(* Logix 5000 project; controller cal1615 1756-L62 rev 20.11; software revision 20.05; part 29 of 82 *)
(* tags used below, declared in another part *)
   FAULT : BOOL;   // Fault AFI
   HMI : BOOL;   // AFI HMI
   p01_sys_scp : SYS_SCP;   // System Scaling
   p01r02 : routine;   // System Misc Control
   p01r09_pb_global_reset : BOOL;   // System Modes PB: Global Fault Reset
   p13_ai_exhaust_amps : REAL;   // Zone 3 Analog Input Exhaust Fan Amps
   p13_ai_exhaust_hz : REAL;   // Zone 3 Analog Input Exhaust Fan HZ
   p13_ai_exhaust_hz_max : REAL;   // Zone 3 Analog Input Exhaust Fan Max HZ
   p13_ai_exhaust_rpm : REAL;   // Zone 3 Analog Input Exhaust Fan RPM
   p13_ai_recirc_amps : REAL;   // Zone 3 Analog Input Recirc Fan Amps
   p13_ai_recirc_hz : REAL;   // Zone 3 Analog Input Supply Fan HZ
   p13_ai_recirc_hz_max : REAL;   // Zone 3 Analog Input Supply Fan max HZ
   p13_ai_recirc_rpm : REAL;   // Zone 3 Analog Input Recirc Fan RPM
   p13_ai_tc01 : REAL;   // Zone 3 Analog Input Control Thermocouple 1
   p13_ai_tc02 : REAL;   // Zone 3 Analog Input Control Thermocouple 2
   p13_ao_cv : REAL;   // Zone 3 Analog Output Control Valve
   p13_ao_exhaust_selected_speed : REAL;   // Zone 3 Analog Output Exhaust Fan VFD Selected Speed
   p13_ao_recirc_selected_speed : REAL;   // Zone 3 Analog Output Recirc Fan VFD Selected Speed
   p13_di_door_open : BOOL;   // Zone 3 Digital Input Access Door Open
   p13_di_exh : acs800_di_normal;   // Zone 3 Digital Inputs Exhaust Fan
   p13_di_exh_fan_mtr_ts : BOOL;   // Zone 3 Digital Input Exhaust Fan Motor Thermostat OK
   p13_di_exh_flow_ok : BOOL;   // Zone 3 Digital Input Exhaust Flow OK
   p13_di_filter_clean : BOOL;   // Zone 3 Digital Input Filter Dirty
   p13_di_recirc : acs800_di_normal;   // Zone 3 Digital Inputs Recirc Fan
   p13_di_recirc_fan_mtr_ts : BOOL;   // Zone 3 Digital Input Recirc Fan Motor Thermostat OK
   p13_di_recirc_flow_ok : BOOL;   // Zone 3 Digital Input Recirc Flow OK
   p13_di_tc01_bo : BOOL;   // Zone 3 Digital Input Control Thermocouple 1 Failure
   p13_di_tc02_bo : BOOL;   // Zone 3 Digital Input Control Thermocouple 2 Failure
   p13_dint_to_hmi : DINT[16];   // Zone 3 Temperature Control VFDs On
   p13_do_exh : acs800_do_normal;   // Zone 3 Digital Output Exhaust Fan
   p13_do_recirc : acs800_do_normal;   // Zone 3 Digital Outputs Supply Fan
   p13_exhaust_input_max : REAL;
   p13_exhaust_input_min : REAL;
   p13_exhaust_output_max : REAL;
   p13_exhaust_output_min : REAL;
   p13_hc_input_max : REAL;
   p13_hc_input_min : REAL;
   p13_hc_output_max : REAL;
   p13_hc_output_min : REAL;
   p13_param_tc01z : REAL;   // Zone 3 Parameter Process Temperature Zero Offset
   p13_param_tc02z : REAL;   // Zone 3 Parameter SupplyTemperature Zero Offset
   p13_recirc_input_max : REAL;
   p13_recirc_input_min : REAL;
   p13_recirc_output_max : REAL;
   p13_recirc_output_min : REAL;
   p13r01 : routine;   // Zone 3 Main
   p13r03 : routine;   // Zone 3 Input
   p13r03_hz : SYS_SCP;   // Zone 3 Analog Inputs SCP Hz
   p13r03_timer_fault : TIMER[4];   // Zone 3 Input Fault Delay
   p13r03_timer_warning : TIMER[4];   // Zone 3 Input Warning Delay
   p13r04 : routine;   // Zone 3 Output
   p13r04_timer_fault : TIMER[4];   // Zone 3 Output Fault Delay
   p13r04_timer_warning : TIMER[4];   // Zone 3 Output Warning Delay
   p13r05 : routine;   // Zone 3 Dint to HMI
   p13r05_exh_status : DINT;
   p13r05_temp_ctl_status : DINT;
   p13r20_state : DINT;   // Zone 3 Temperature Control State
   p13r20_status : DINT;   // Zone 3 Temperature Control Sequence Status
   p13r30 : routine;   // Zone 3 Temperature Control
   p13r30_permissive_run : BOOL;   // Zone 3 Temperature Control Run Permissive
   p13r30_request_cool : BOOL;   // Zone 3 Temperature Control Request Cooling
   p13r30_request_manual : BOOL;   // Zone 3 Temperature Control Request Manual Control
   p13r30_vfds_ready : BOOL;   // Zone 3 Temperature Control VFDs On
   p13r31 : routine;   // Zone 3 Exhaust VFD
   p13r31_request_auto_run : BOOL;   // Zone 3 Exhaust Fan Run Request
   p13r31_request_auto_stop : BOOL;   // Zone 3 Exhaust VFD Request Auto Stop
   p13r31_vfd_stopped : BOOL;   // Zone 3 Exhaust VFD VFD Stopped
   p13r32_request_auto_run : BOOL;   // Zone 3 Recirc Fan Run Request
   p13r32_request_auto_stop : BOOL;   // Zone 3 Recirc VFD Request Auto Stop
(* P13_Zone_3, continued *)

ROUTINE R03_Input   (* ladder *)
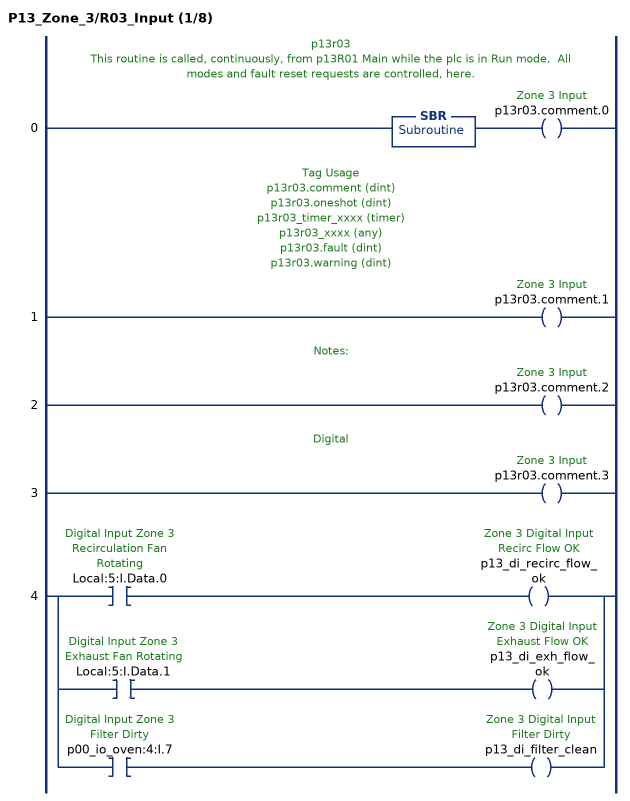
   // p13r03
   // This routine is called, continuously, from p13R01 Main while the plc is in Run mode.  All modes and fault reset requests are controlled, here.
   0: SBR()OTE(p13r03.comment.0);
   // Tag Usage
   // p13r03.comment (dint)
   // p13r03.oneshot (dint)
   // p13r03_timer_xxxx (timer)
   // p13r03_xxxx (any)
   // p13r03.fault (dint)
   // p13r03.warning (dint)
   1: OTE(p13r03.comment.1);
   // Notes:
   2: OTE(p13r03.comment.2);
   // Digital
   3: OTE(p13r03.comment.3);
   4: [XIC(Local:5:I.Data.0) OTE(p13_di_recirc_flow_ok) ,XIC(Local:5:I.Data.1) OTE(p13_di_exh_flow_ok) ,XIC(p00_io_oven:4:I.7) OTE(p13_di_filter_clean) ];
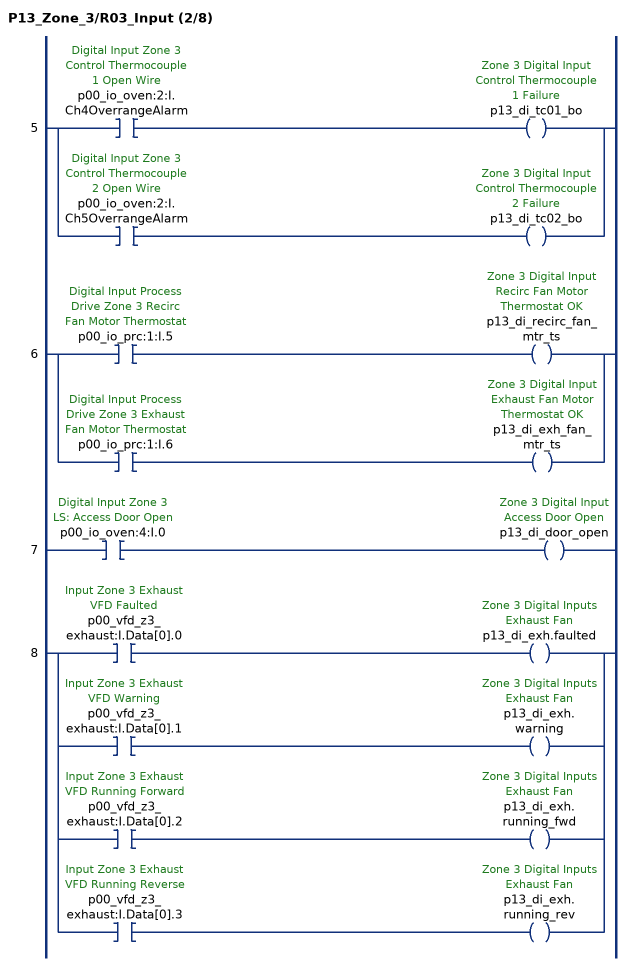
   5: [XIC(p00_io_oven:2:I.Ch4OverrangeAlarm) OTE(p13_di_tc01_bo) ,XIC(p00_io_oven:2:I.Ch5OverrangeAlarm) OTE(p13_di_tc02_bo) ];
   6: [XIC(p00_io_prc:1:I.5) OTE(p13_di_recirc_fan_mtr_ts) ,XIC(p00_io_prc:1:I.6) OTE(p13_di_exh_fan_mtr_ts) ];
   7: XIC(p00_io_oven:4:I.0)OTE(p13_di_door_open);
   8: [XIC(p00_vfd_z3_exhaust:I.Data[0].0) OTE(p13_di_exh.faulted) ,XIC(p00_vfd_z3_exhaust:I.Data[0].1) OTE(p13_di_exh.warning) ,XIC(p00_vfd_z3_exhaust:I.Data[0].2) OTE(p13_di_exh.running_fwd) ,XIC(p00_vfd_z3_exhaust:I.Data[0].3) OTE(p13_di_exh.running_rev) ];
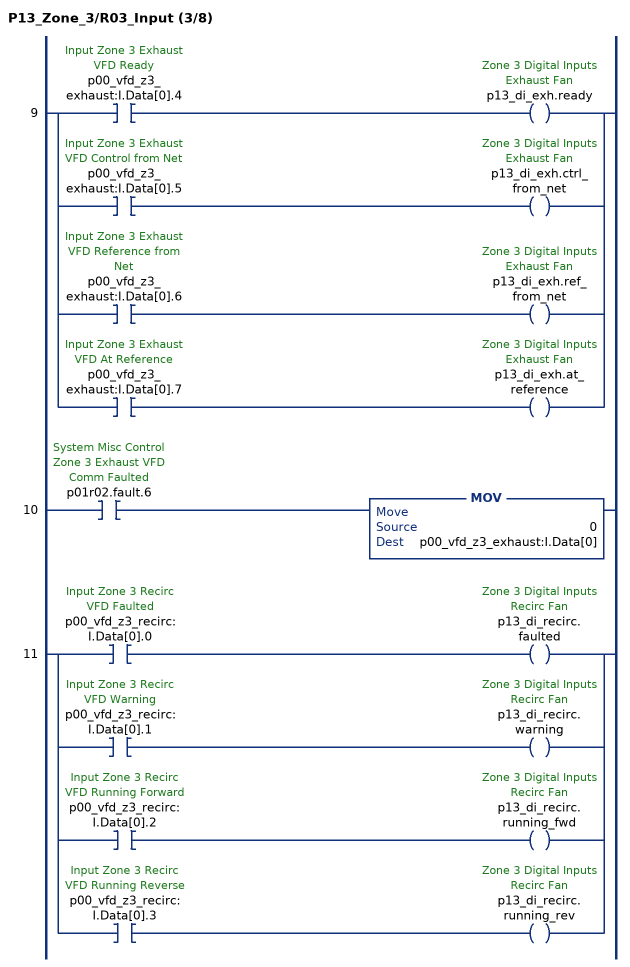
   9: [XIC(p00_vfd_z3_exhaust:I.Data[0].4) OTE(p13_di_exh.ready) ,XIC(p00_vfd_z3_exhaust:I.Data[0].5) OTE(p13_di_exh.ctrl_from_net) ,XIC(p00_vfd_z3_exhaust:I.Data[0].6) OTE(p13_di_exh.ref_from_net) ,XIC(p00_vfd_z3_exhaust:I.Data[0].7) OTE(p13_di_exh.at_reference) ];
   10: XIC(p01r02.fault.6)MOV(0,p00_vfd_z3_exhaust:I.Data[0]);
   11: [XIC(p00_vfd_z3_recirc:I.Data[0].0) OTE(p13_di_recirc.faulted) ,XIC(p00_vfd_z3_recirc:I.Data[0].1) OTE(p13_di_recirc.warning) ,XIC(p00_vfd_z3_recirc:I.Data[0].2) OTE(p13_di_recirc.running_fwd) ,XIC(p00_vfd_z3_recirc:I.Data[0].3) OTE(p13_di_recirc.running_rev) ];
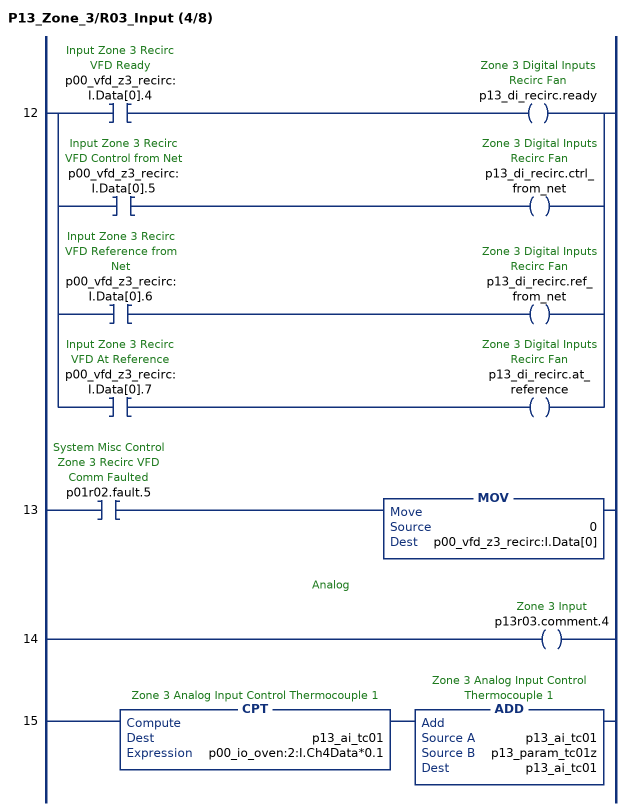
   12: [XIC(p00_vfd_z3_recirc:I.Data[0].4) OTE(p13_di_recirc.ready) ,XIC(p00_vfd_z3_recirc:I.Data[0].5) OTE(p13_di_recirc.ctrl_from_net) ,XIC(p00_vfd_z3_recirc:I.Data[0].6) OTE(p13_di_recirc.ref_from_net) ,XIC(p00_vfd_z3_recirc:I.Data[0].7) OTE(p13_di_recirc.at_reference) ];
   13: XIC(p01r02.fault.5)MOV(0,p00_vfd_z3_recirc:I.Data[0]);
   // Analog
   14: OTE(p13r03.comment.4);
   15: CPT(p13_ai_tc01,p00_io_oven:2:I.Ch4Data*0.1)ADD(p13_ai_tc01,p13_param_tc01z,p13_ai_tc01);
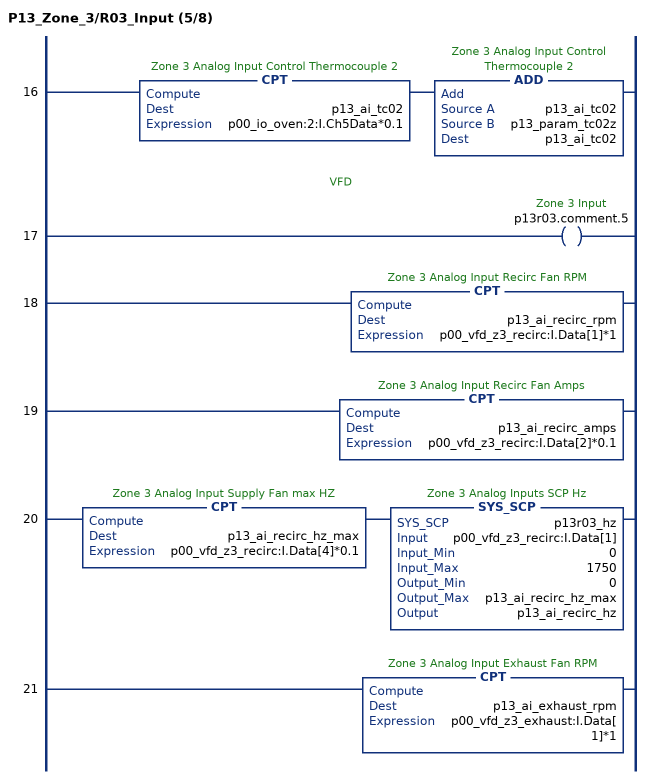
   16: CPT(p13_ai_tc02,p00_io_oven:2:I.Ch5Data*0.1)ADD(p13_ai_tc02,p13_param_tc02z,p13_ai_tc02);
   // VFD
   17: OTE(p13r03.comment.5);
   18: CPT(p13_ai_recirc_rpm,p00_vfd_z3_recirc:I.Data[1]*1);
   19: CPT(p13_ai_recirc_amps,p00_vfd_z3_recirc:I.Data[2]*0.1);
   20: CPT(p13_ai_recirc_hz_max,p00_vfd_z3_recirc:I.Data[4]*0.1)SYS_SCP(p13r03_hz,p00_vfd_z3_recirc:I.Data[1],0,1750,0,p13_ai_recirc_hz_max,p13_ai_recirc_hz);
   21: CPT(p13_ai_exhaust_rpm,p00_vfd_z3_exhaust:I.Data[1]*1);
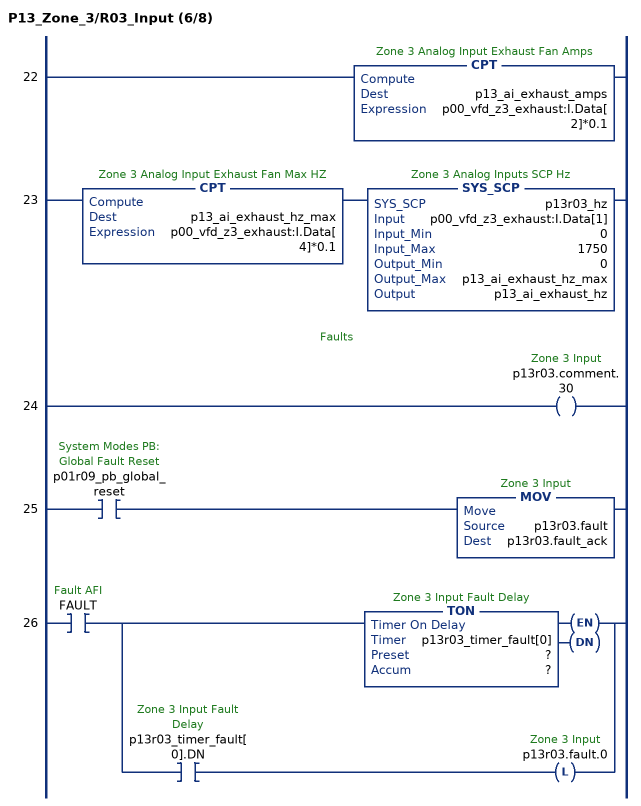
   22: CPT(p13_ai_exhaust_amps,p00_vfd_z3_exhaust:I.Data[2]*0.1);
   23: CPT(p13_ai_exhaust_hz_max,p00_vfd_z3_exhaust:I.Data[4]*0.1)SYS_SCP(p13r03_hz,p00_vfd_z3_exhaust:I.Data[1],0,1750,0,p13_ai_exhaust_hz_max,p13_ai_exhaust_hz);
   // Faults
   24: OTE(p13r03.comment.30);
   25: XIC(p01r09_pb_global_reset)MOV(p13r03.fault,p13r03.fault_ack);
   26: XIC(FAULT)[TON(p13r03_timer_fault[0],?,?) ,XIC(p13r03_timer_fault[0].DN) OTL(p13r03.fault.0) ];
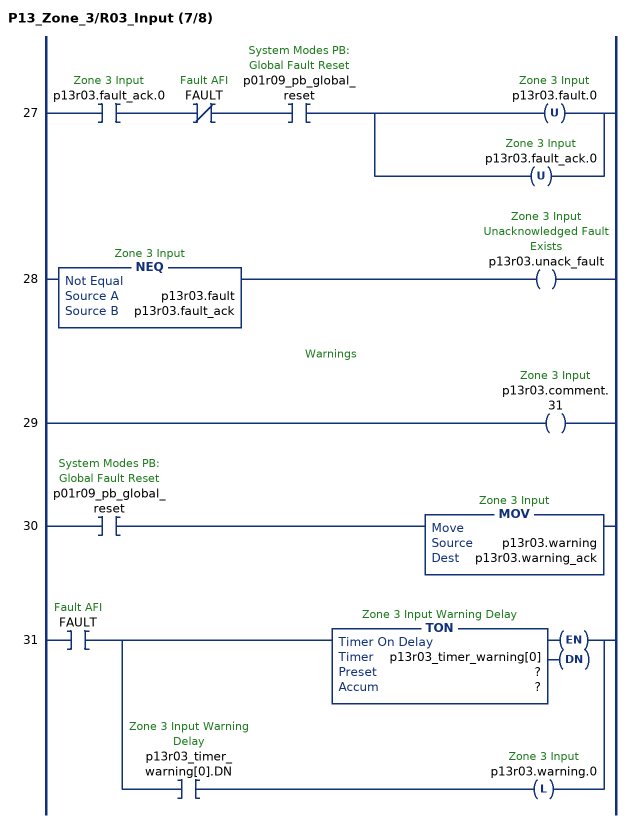
   27: XIC(p13r03.fault_ack.0)XIO(FAULT)XIC(p01r09_pb_global_reset)[OTU(p13r03.fault.0) ,OTU(p13r03.fault_ack.0) ];
   28: NEQ(p13r03.fault,p13r03.fault_ack)OTE(p13r03.unack_fault);
   // Warnings
   29: OTE(p13r03.comment.31);
   30: XIC(p01r09_pb_global_reset)MOV(p13r03.warning,p13r03.warning_ack);
   31: XIC(FAULT)[TON(p13r03_timer_warning[0],?,?) ,XIC(p13r03_timer_warning[0].DN) OTL(p13r03.warning.0) ];
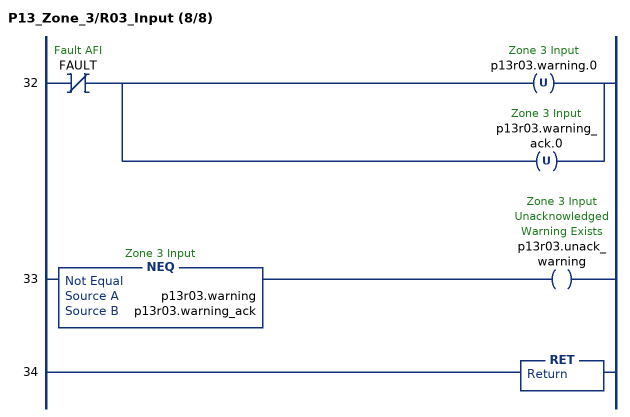
   32: XIO(FAULT)[OTU(p13r03.warning.0) ,OTU(p13r03.warning_ack.0) ];
   33: NEQ(p13r03.warning,p13r03.warning_ack)OTE(p13r03.unack_warning);
   34: RET();
END_ROUTINE

ROUTINE R04_Output   (* ladder *)
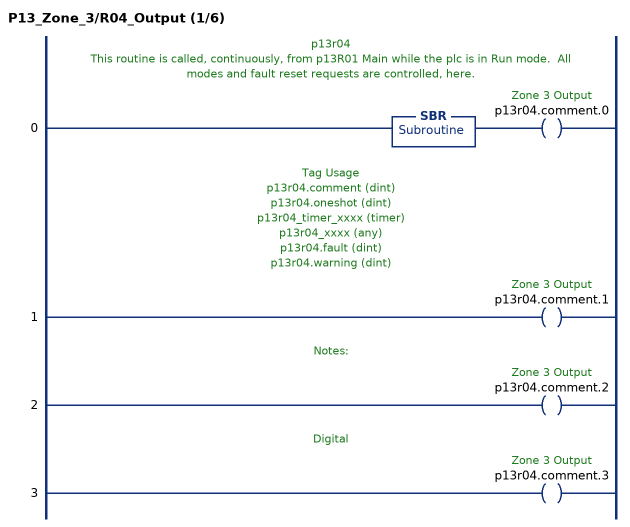
   // p13r04
   // This routine is called, continuously, from p13R01 Main while the plc is in Run mode.  All modes and fault reset requests are controlled, here.
   0: SBR()OTE(p13r04.comment.0);
   // Tag Usage
   // p13r04.comment (dint)
   // p13r04.oneshot (dint)
   // p13r04_timer_xxxx (timer)
   // p13r04_xxxx (any)
   // p13r04.fault (dint)
   // p13r04.warning (dint)
   1: OTE(p13r04.comment.1);
   // Notes:
   2: OTE(p13r04.comment.2);
   // Digital
   3: OTE(p13r04.comment.3);
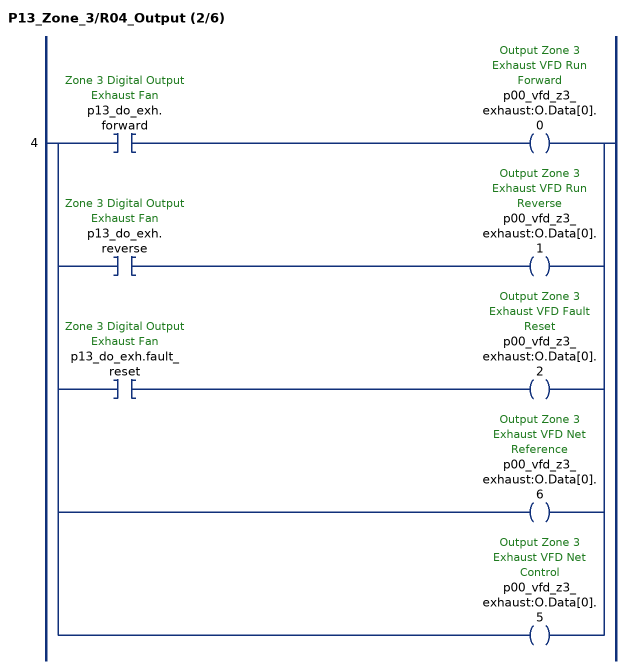
   4: [XIC(p13_do_exh.forward) OTE(p00_vfd_z3_exhaust:O.Data[0].0) ,XIC(p13_do_exh.reverse) OTE(p00_vfd_z3_exhaust:O.Data[0].1) ,XIC(p13_do_exh.fault_reset) OTE(p00_vfd_z3_exhaust:O.Data[0].2) ,OTE(p00_vfd_z3_exhaust:O.Data[0].6) ,OTE(p00_vfd_z3_exhaust:O.Data[0].5) ];
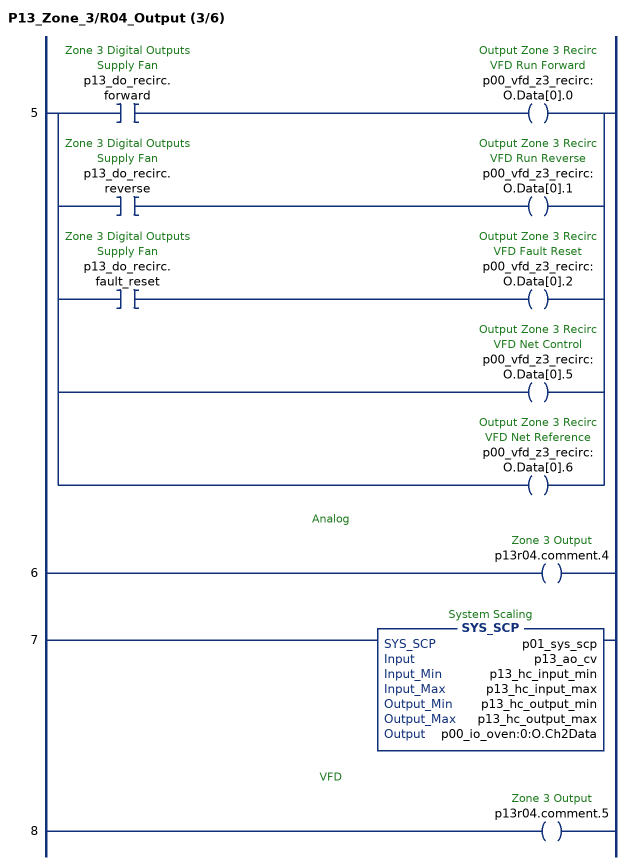
   5: [XIC(p13_do_recirc.forward) OTE(p00_vfd_z3_recirc:O.Data[0].0) ,XIC(p13_do_recirc.reverse) OTE(p00_vfd_z3_recirc:O.Data[0].1) ,XIC(p13_do_recirc.fault_reset) OTE(p00_vfd_z3_recirc:O.Data[0].2) ,OTE(p00_vfd_z3_recirc:O.Data[0].5) ,OTE(p00_vfd_z3_recirc:O.Data[0].6) ];
   // Analog
   6: OTE(p13r04.comment.4);
   7: SYS_SCP(p01_sys_scp,p13_ao_cv,p13_hc_input_min,p13_hc_input_max,p13_hc_output_min,p13_hc_output_max,p00_io_oven:0:O.Ch2Data);
   // VFD
   8: OTE(p13r04.comment.5);
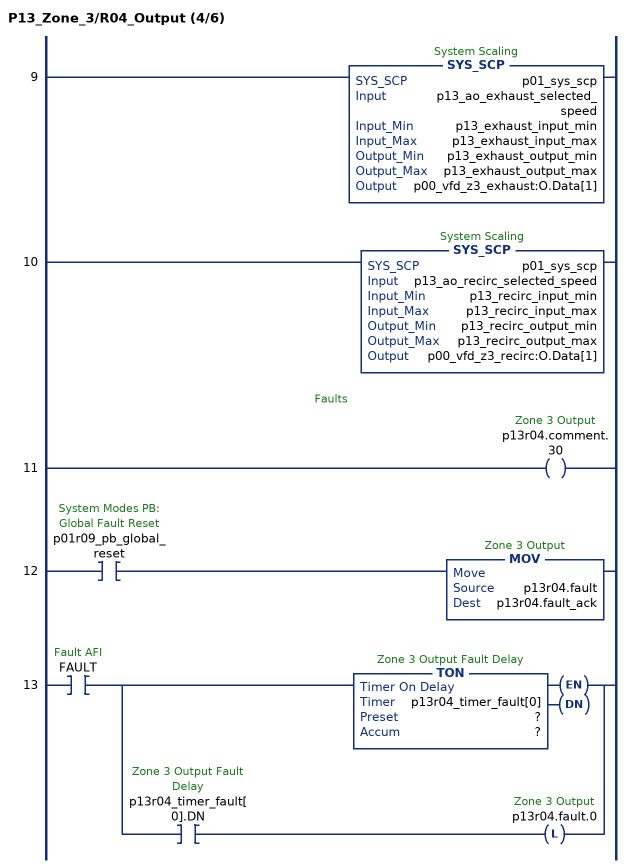
   9: SYS_SCP(p01_sys_scp,p13_ao_exhaust_selected_speed,p13_exhaust_input_min,p13_exhaust_input_max,p13_exhaust_output_min,p13_exhaust_output_max,p00_vfd_z3_exhaust:O.Data[1]);
   10: SYS_SCP(p01_sys_scp,p13_ao_recirc_selected_speed,p13_recirc_input_min,p13_recirc_input_max,p13_recirc_output_min,p13_recirc_output_max,p00_vfd_z3_recirc:O.Data[1]);
   // Faults
   11: OTE(p13r04.comment.30);
   12: XIC(p01r09_pb_global_reset)MOV(p13r04.fault,p13r04.fault_ack);
   13: XIC(FAULT)[TON(p13r04_timer_fault[0],?,?) ,XIC(p13r04_timer_fault[0].DN) OTL(p13r04.fault.0) ];
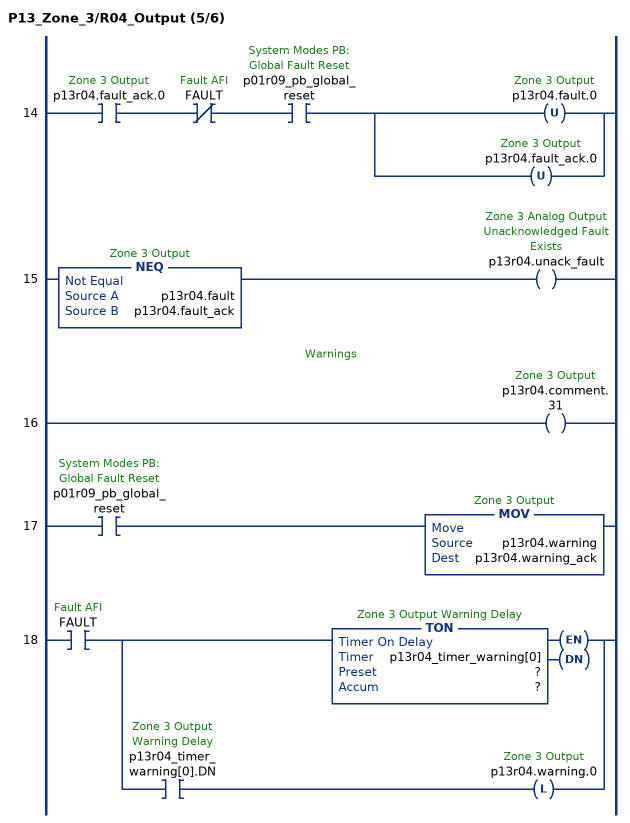
   14: XIC(p13r04.fault_ack.0)XIO(FAULT)XIC(p01r09_pb_global_reset)[OTU(p13r04.fault.0) ,OTU(p13r04.fault_ack.0) ];
   15: NEQ(p13r04.fault,p13r04.fault_ack)OTE(p13r04.unack_fault);
   // Warnings
   16: OTE(p13r04.comment.31);
   17: XIC(p01r09_pb_global_reset)MOV(p13r04.warning,p13r04.warning_ack);
   18: XIC(FAULT)[TON(p13r04_timer_warning[0],?,?) ,XIC(p13r04_timer_warning[0].DN) OTL(p13r04.warning.0) ];
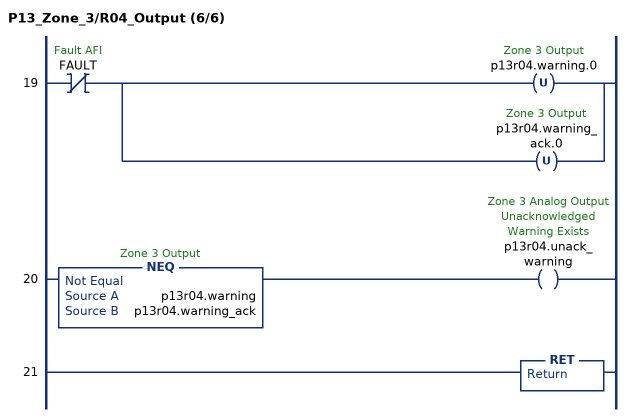
   19: XIO(FAULT)[OTU(p13r04.warning.0) ,OTU(p13r04.warning_ack.0) ];
   20: NEQ(p13r04.warning,p13r04.warning_ack)OTE(p13r04.unack_warning);
   21: RET();
END_ROUTINE

ROUTINE R05_Dint_to_HMI   (* ladder *)
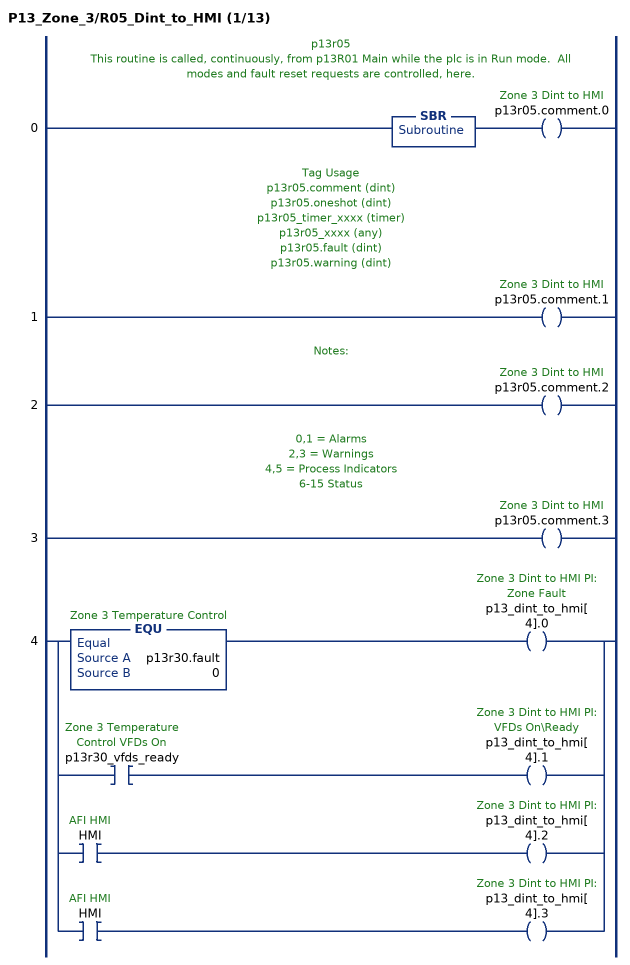
   // p13r05
   // This routine is called, continuously, from p13R01 Main while the plc is in Run mode.  All modes and fault reset requests are controlled, here.
   0: SBR()OTE(p13r05.comment.0);
   // Tag Usage
   // p13r05.comment (dint)
   // p13r05.oneshot (dint)
   // p13r05_timer_xxxx (timer)
   // p13r05_xxxx (any)
   // p13r05.fault (dint)
   // p13r05.warning (dint)
   1: OTE(p13r05.comment.1);
   // Notes:
   2: OTE(p13r05.comment.2);
   // 0,1 = Alarms
   // 2,3 = Warnings
   // 4,5 = Process Indicators
   // 6-15 Status
   3: OTE(p13r05.comment.3);
   4: [EQU(p13r30.fault,0) OTE(p13_dint_to_hmi[4].0) ,XIC(p13r30_vfds_ready) OTE(p13_dint_to_hmi[4].1) ,XIC(HMI) OTE(p13_dint_to_hmi[4].2) ,XIC(HMI) OTE(p13_dint_to_hmi[4].3) ];
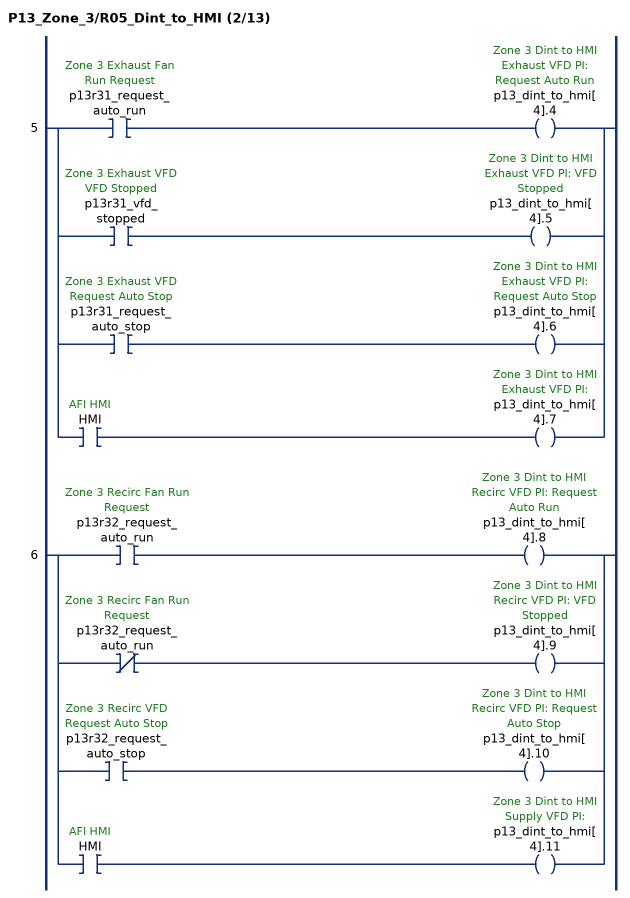
   5: [XIC(p13r31_request_auto_run) OTE(p13_dint_to_hmi[4].4) ,XIC(p13r31_vfd_stopped) OTE(p13_dint_to_hmi[4].5) ,XIC(p13r31_request_auto_stop) OTE(p13_dint_to_hmi[4].6) ,XIC(HMI) OTE(p13_dint_to_hmi[4].7) ];
   6: [XIC(p13r32_request_auto_run) OTE(p13_dint_to_hmi[4].8) ,XIO(p13r32_request_auto_run) OTE(p13_dint_to_hmi[4].9) ,XIC(p13r32_request_auto_stop) OTE(p13_dint_to_hmi[4].10) ,XIC(HMI) OTE(p13_dint_to_hmi[4].11) ];
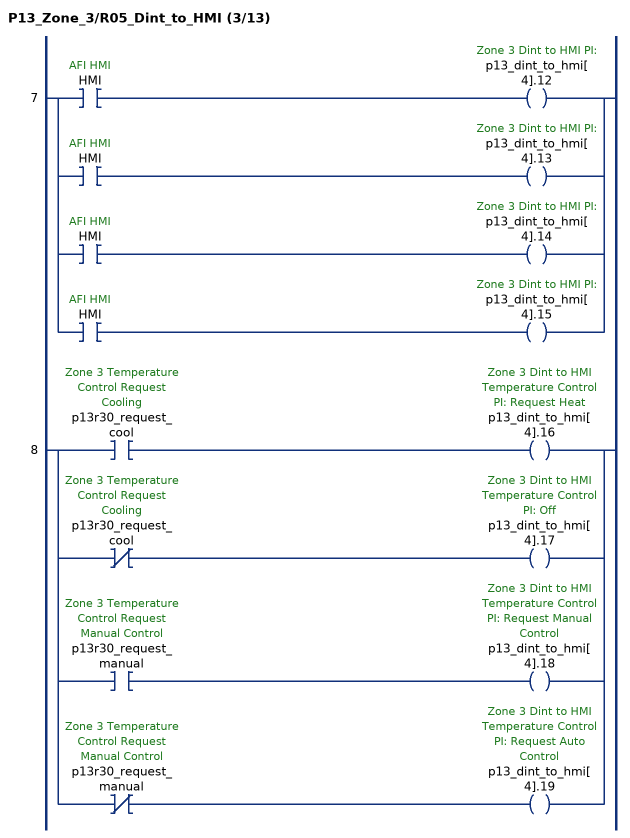
   7: [XIC(HMI) OTE(p13_dint_to_hmi[4].12) ,XIC(HMI) OTE(p13_dint_to_hmi[4].13) ,XIC(HMI) OTE(p13_dint_to_hmi[4].14) ,XIC(HMI) OTE(p13_dint_to_hmi[4].15) ];
   8: [XIC(p13r30_request_cool) OTE(p13_dint_to_hmi[4].16) ,XIO(p13r30_request_cool) OTE(p13_dint_to_hmi[4].17) ,XIC(p13r30_request_manual) OTE(p13_dint_to_hmi[4].18) ,XIO(p13r30_request_manual) OTE(p13_dint_to_hmi[4].19) ];
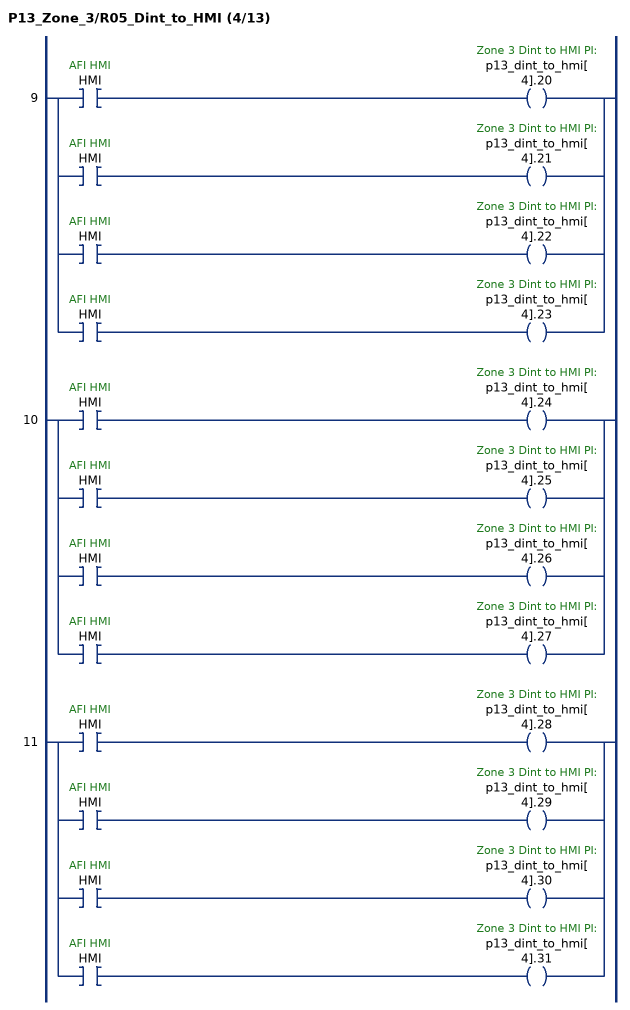
   9: [XIC(HMI) OTE(p13_dint_to_hmi[4].20) ,XIC(HMI) OTE(p13_dint_to_hmi[4].21) ,XIC(HMI) OTE(p13_dint_to_hmi[4].22) ,XIC(HMI) OTE(p13_dint_to_hmi[4].23) ];
   10: [XIC(HMI) OTE(p13_dint_to_hmi[4].24) ,XIC(HMI) OTE(p13_dint_to_hmi[4].25) ,XIC(HMI) OTE(p13_dint_to_hmi[4].26) ,XIC(HMI) OTE(p13_dint_to_hmi[4].27) ];
   11: [XIC(HMI) OTE(p13_dint_to_hmi[4].28) ,XIC(HMI) OTE(p13_dint_to_hmi[4].29) ,XIC(HMI) OTE(p13_dint_to_hmi[4].30) ,XIC(HMI) OTE(p13_dint_to_hmi[4].31) ];
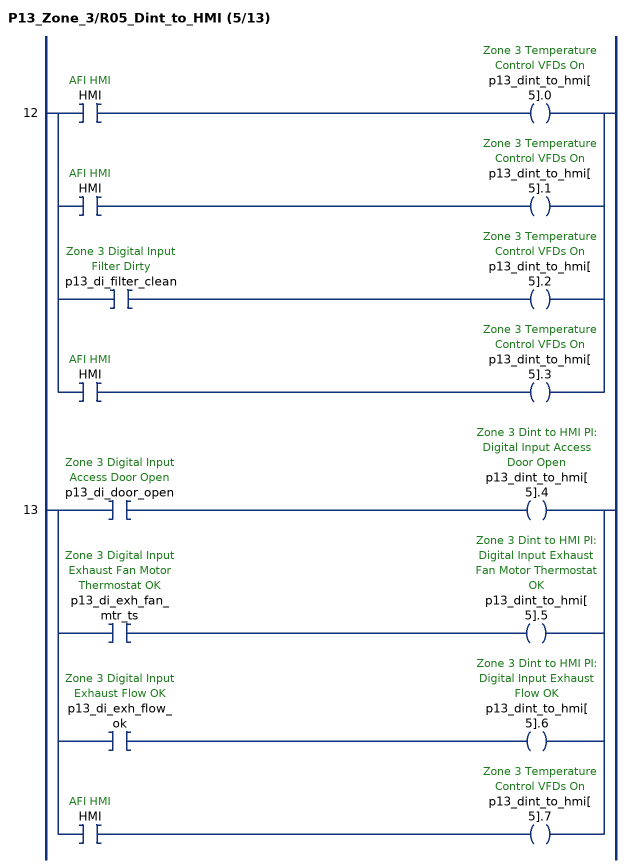
   12: [XIC(HMI) OTE(p13_dint_to_hmi[5].0) ,XIC(HMI) OTE(p13_dint_to_hmi[5].1) ,XIC(p13_di_filter_clean) OTE(p13_dint_to_hmi[5].2) ,XIC(HMI) OTE(p13_dint_to_hmi[5].3) ];
   13: [XIC(p13_di_door_open) OTE(p13_dint_to_hmi[5].4) ,XIC(p13_di_exh_fan_mtr_ts) OTE(p13_dint_to_hmi[5].5) ,XIC(p13_di_exh_flow_ok) OTE(p13_dint_to_hmi[5].6) ,XIC(HMI) OTE(p13_dint_to_hmi[5].7) ];
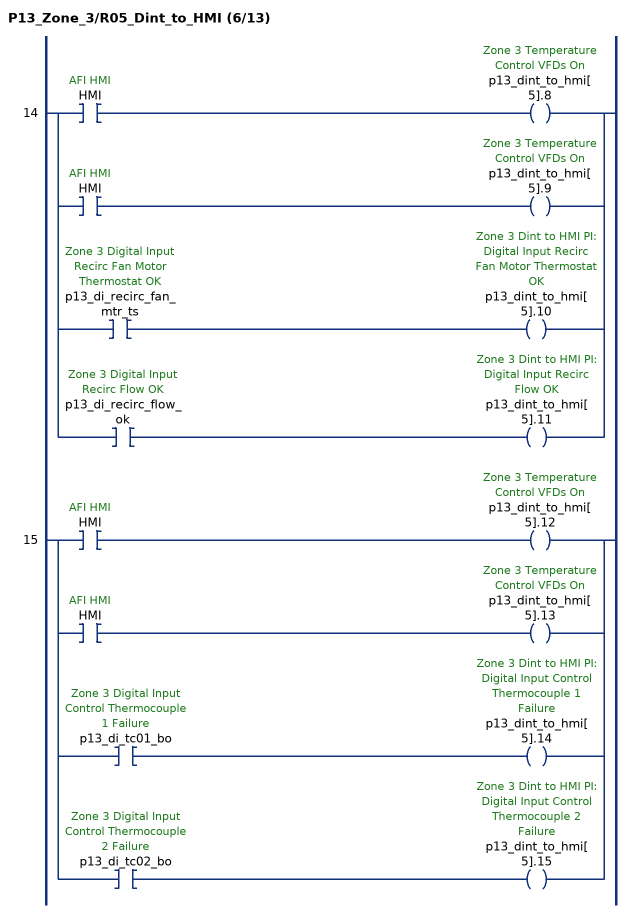
   14: [XIC(HMI) OTE(p13_dint_to_hmi[5].8) ,XIC(HMI) OTE(p13_dint_to_hmi[5].9) ,XIC(p13_di_recirc_fan_mtr_ts) OTE(p13_dint_to_hmi[5].10) ,XIC(p13_di_recirc_flow_ok) OTE(p13_dint_to_hmi[5].11) ];
   15: [XIC(HMI) OTE(p13_dint_to_hmi[5].12) ,XIC(HMI) OTE(p13_dint_to_hmi[5].13) ,XIC(p13_di_tc01_bo) OTE(p13_dint_to_hmi[5].14) ,XIC(p13_di_tc02_bo) OTE(p13_dint_to_hmi[5].15) ];
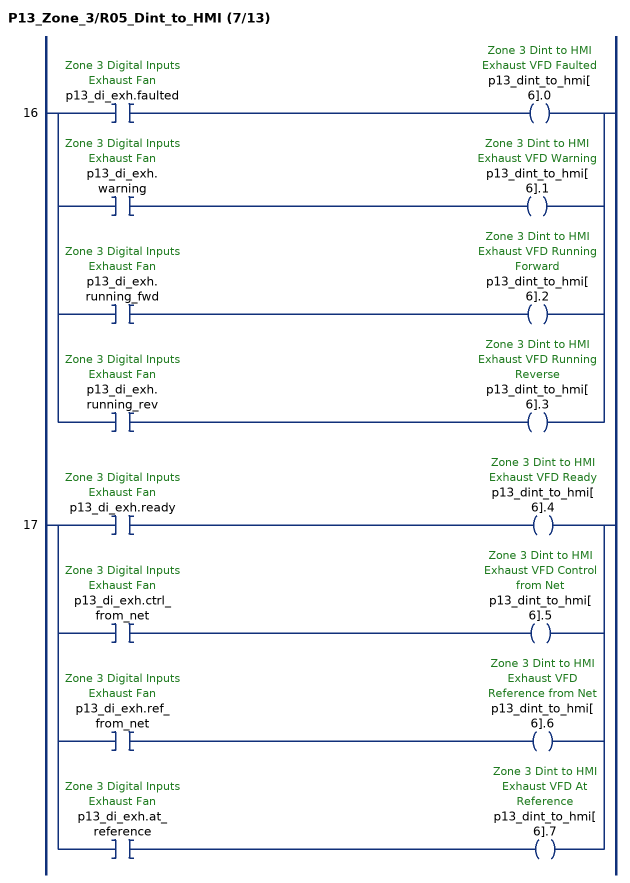
   16: [XIC(p13_di_exh.faulted) OTE(p13_dint_to_hmi[6].0) ,XIC(p13_di_exh.warning) OTE(p13_dint_to_hmi[6].1) ,XIC(p13_di_exh.running_fwd) OTE(p13_dint_to_hmi[6].2) ,XIC(p13_di_exh.running_rev) OTE(p13_dint_to_hmi[6].3) ];
   17: [XIC(p13_di_exh.ready) OTE(p13_dint_to_hmi[6].4) ,XIC(p13_di_exh.ctrl_from_net) OTE(p13_dint_to_hmi[6].5) ,XIC(p13_di_exh.ref_from_net) OTE(p13_dint_to_hmi[6].6) ,XIC(p13_di_exh.at_reference) OTE(p13_dint_to_hmi[6].7) ];
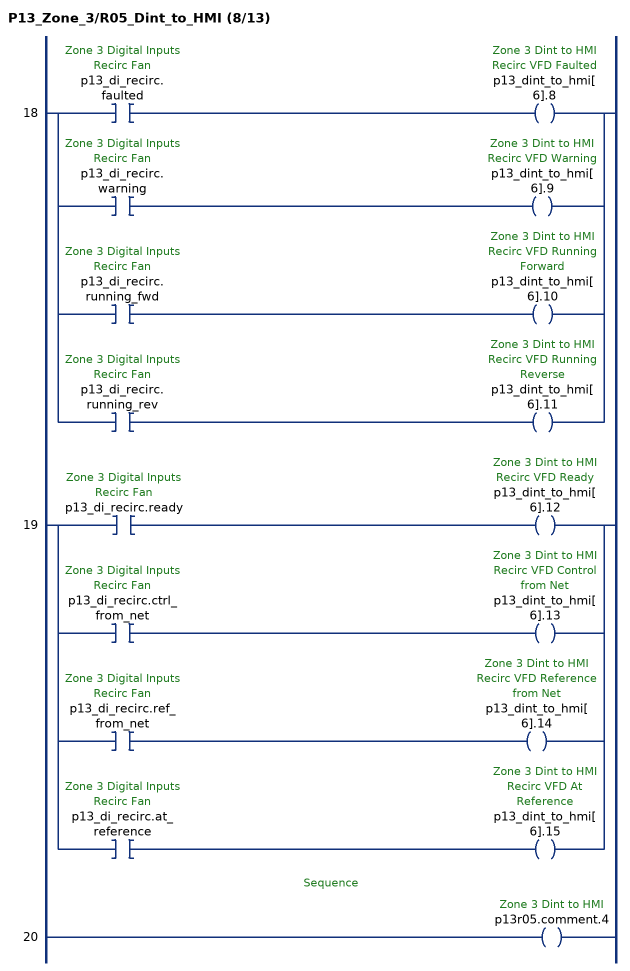
   18: [XIC(p13_di_recirc.faulted) OTE(p13_dint_to_hmi[6].8) ,XIC(p13_di_recirc.warning) OTE(p13_dint_to_hmi[6].9) ,XIC(p13_di_recirc.running_fwd) OTE(p13_dint_to_hmi[6].10) ,XIC(p13_di_recirc.running_rev) OTE(p13_dint_to_hmi[6].11) ];
   19: [XIC(p13_di_recirc.ready) OTE(p13_dint_to_hmi[6].12) ,XIC(p13_di_recirc.ctrl_from_net) OTE(p13_dint_to_hmi[6].13) ,XIC(p13_di_recirc.ref_from_net) OTE(p13_dint_to_hmi[6].14) ,XIC(p13_di_recirc.at_reference) OTE(p13_dint_to_hmi[6].15) ];
   // Sequence
   20: OTE(p13r05.comment.4);
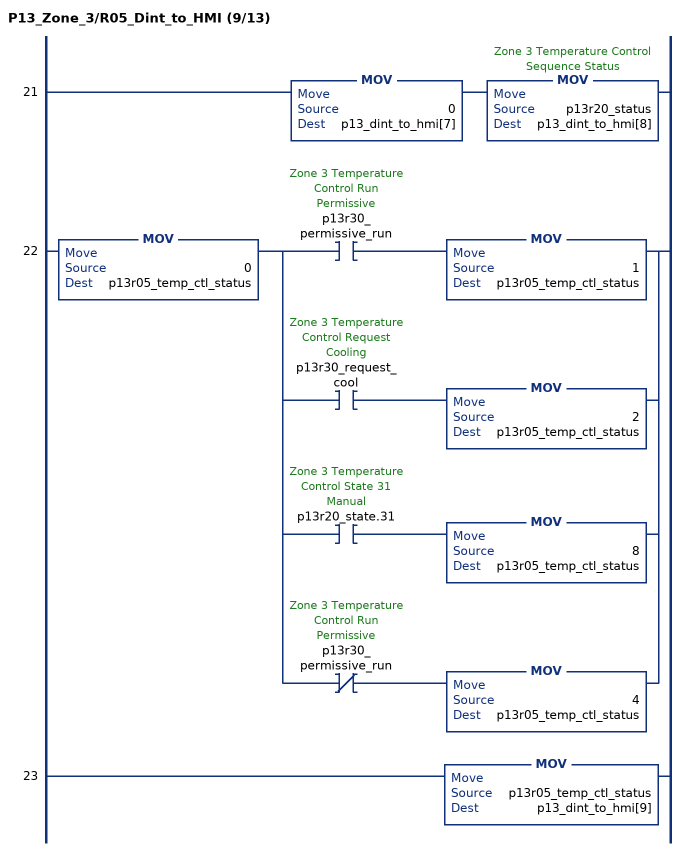
   21: MOV(0,p13_dint_to_hmi[7])MOV(p13r20_status,p13_dint_to_hmi[8]);
   22: MOV(0,p13r05_temp_ctl_status)[XIC(p13r30_permissive_run) MOV(1,p13r05_temp_ctl_status) ,XIC(p13r30_request_cool) MOV(2,p13r05_temp_ctl_status) ,XIC(p13r20_state.31) MOV(8,p13r05_temp_ctl_status) ,XIO(p13r30_permissive_run) MOV(4,p13r05_temp_ctl_status) ];
   23: MOV(p13r05_temp_ctl_status,p13_dint_to_hmi[9]);
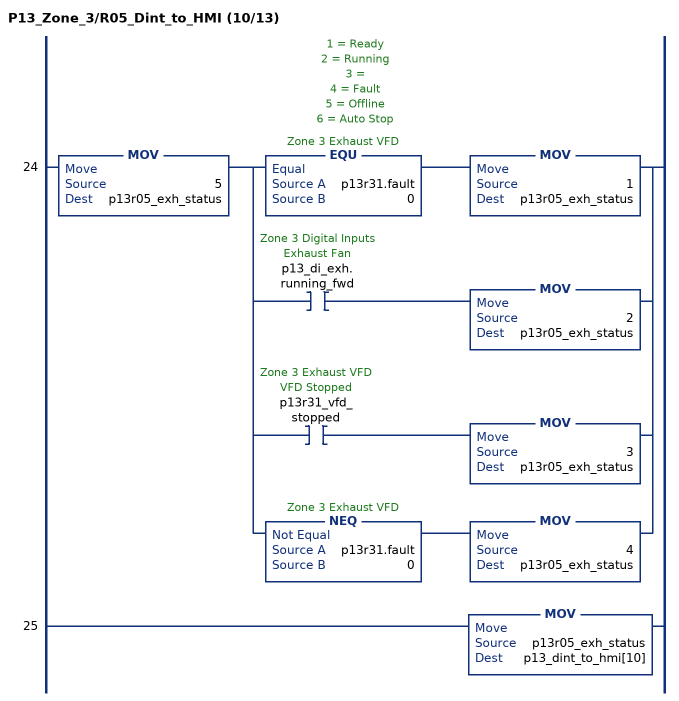
   // 1 = Ready
   // 2 = Running
   // 3 =
   // 4 = Fault
   // 5 = Offline
   // 6 = Auto Stop
   24: MOV(5,p13r05_exh_status)[EQU(p13r31.fault,0) MOV(1,p13r05_exh_status) ,XIC(p13_di_exh.running_fwd) MOV(2,p13r05_exh_status) ,XIC(p13r31_vfd_stopped) MOV(3,p13r05_exh_status) ,NEQ(p13r31.fault,0) MOV(4,p13r05_exh_status) ];
   25: MOV(p13r05_exh_status,p13_dint_to_hmi[10]);
